// TwinCAT 3 PLC project Plc
// ProgramVersion: 3.1.4024.0
// libraries:
//   Tc2_Standard, * (Beckhoff Automation GmbH)
//   Tc2_System, * (Beckhoff Automation GmbH)
//   Tc3_Module, * (Beckhoff Automation GmbH)
//   VisuSymbols,3.5.10.0,System
// project tree:
//   / Gestore di visualizzazione.TcVMO (not stored), GlobalTextList.TcGTLO, PlcTask.TcTTO
//   POUs/ MAIN.TcPOU
//   VISUs/ Visualization.TcVIS
// real-time tasks:
//   TASK PlcTask: cycle T#10ms, priority 20, ADS port 350

CONFIGURATION Plc
    RESOURCE PLC ON TwinCAT3
        TASK PlcTask(INTERVAL := T#10ms, PRIORITY := 20);
        PROGRAM MAIN WITH PlcTask : MAIN;
    END_RESOURCE
END_CONFIGURATION

// ---- POUs/MAIN.TcPOU
PROGRAM MAIN
VAR
	Verde: BOOL;
	Giallo: BOOL;
	Rosso: BOOL;
	Ton1: TON;
	Ton2: TON;
	Ton3: TON;
END_VAR

Ton1(IN:= NOT Ton3.Q, PT:= T#5S);
Ton2(IN:= Ton1.Q, PT:= T#2S);
Ton3(IN:= Ton2.Q, PT:= T#8S);

Verde:= NOT Ton1.Q;
Giallo:= NOT Ton2.Q AND Ton1.Q;
Rosso:= NOT Ton3.Q AND Ton2.Q;

END_PROGRAM

// ---- VISUs/Visualization.TcVIS
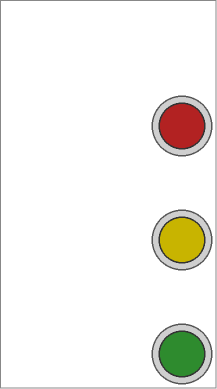
VISUALIZATION Visualization  // 217x389
    Lamp1 (147,91 70x70), variable: MAIN.Rosso, style: Lamp-Lamp1-Red
    Lamp1 (147,205 70x70), variable: MAIN.Giallo, style: Lamp-Lamp1-Yellow
    Lamp1 (147,319 70x70), variable: MAIN.Verde, style: Lamp-Lamp1-Green
END_VISUALIZATION
